// TIA Portal V20 export
TYPE "LER_typeRadiusMeasureControlNode"
// stored: Access Published
   STRUCT
      commands { ExternalWritable := 'False'} : "LER_typeRadiusMeasureCommnads";
      monitoring { ExternalWritable := 'False'} : "LER_typeRadiusMeasureMonitioing";
   END_STRUCT;
END_TYPE
